ADAPTER IPhaseStatus (* Adapter Interface *)
  (* Standard: 61499-1 *)
  (* Version 0.0, 19/04/2022, schneider, Schneider Electric *)
  PACKAGE SE.Nereda;
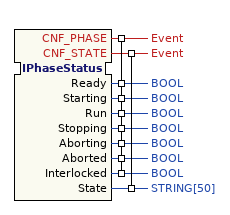
  EVENT_OUTPUT
    CNF_PHASE WITH Interlocked, Ready, Starting, Run, Stopping, Aborting, Aborted;
    CNF_STATE WITH State;
  END_EVENT
  VAR_OUTPUT
    Ready : BOOL;
    Starting : BOOL;
    Run : BOOL;
    Stopping : BOOL;
    Aborting : BOOL;
    Aborted : BOOL;
    Interlocked : BOOL;
    State : STRING[50];
  END_VAR
  SERVICE SOCKET/PLUG
    SEQUENCE request_confirm
      SOCKET.REQ(REQD) -> PLUG.REQ(REQD);
      PLUG.CNF_READY(CNFD) -> SOCKET.CNF_READY(CNFD);
    END_SEQUENCE
    SEQUENCE indication_response
      PLUG.CNF_STARTING(INDD) -> SOCKET.CNF_STARTING(INDD);
      SOCKET.New_Op_Cdt(RSPD) -> PLUG.New_Op_Cdt(RSPD);
    END_SEQUENCE
  END_SERVICE
END_ADAPTER
